// TIA Portal V18 export
VAR_GLOBAL   // PLC tag table "默认变量表"
   Tag_1 AT %M0.0 : Bool;
   Tag_2 AT %M0.1 : Bool;
   Tag_3 AT %M0.2 : Bool;
   Tag_4 AT %M0.3 : Bool;
   Tag_5 AT %M0.4 : Bool;
   Tag_6 AT %M0.5 : Bool;
END_VAR
